{attribute addProperty BoxType "EL6851-0000-0017"}
{attribute addProperty Id "Transmit_acceptedAT %I*BOOL811Receive_toggleAT %I*BOOL812Cyclic_TxD_disabledAT %I*BOOL813Default_data_sentAT %I*BOOL814Frame_sent_toggleAT %I*BOOL8114TxPDO_ToggleAT %I*BOOL819Channel_lengthAT %I*UINT16217Start_codeAT %I*USINT8118"}
{attribute addProperty CRC "3850382601"}
{attribute addProperty SizeInBites "72"}
{attribute addProperty SizeInBytes "9"}
TYPE DMX_Status_E5802D09 :
STRUCT
	{attribute addProperty Name "Transmit_accepted"}
	Transmit_accepted AT %I* : BOOL;
	{attribute addProperty Name "Receive_toggle"}
	Receive_toggle AT %I* : BOOL;
	{attribute addProperty Name "Cyclic_TxD_disabled"}
	Cyclic_TxD_disabled AT %I* : BOOL;
	{attribute addProperty Name "Default_data_sent"}
	Default_data_sent AT %I* : BOOL;
	{attribute addProperty Name "Frame_sent_toggle"}
	Frame_sent_toggle AT %I* : BOOL;
	{attribute addProperty Name "TxPDO_Toggle"}
	TxPDO_Toggle AT %I* : BOOL;
	{attribute addProperty Name "Channel_length"}
	Channel_length AT %I* : UINT;
	{attribute addProperty Name "Start_code"}
	Start_code AT %I* : USINT;
END_STRUCT
END_TYPE

(* stored: Version 1.2.0.0, ProductVersion 3.1.4024.9
   DUT DMX_Status_E5802D09: Id {665e4a63-2c10-4a8d-9459-283397abd407} *)
